FUNCTION_BLOCK FB_Simple
VAR
  boolean:BOOL := TRUE;
END_VAR

// No code here

END_FUNCTION_BLOCK

(* stored: Version 1.1.0.1, ProductVersion 3.1.4024.3
   POU FB_Simple: Id {7b81e162-46f6-4a08-85f1-6c0ae9b32d13}, SpecialFunc None *)
